// TIA Portal V15.1 export
FUNCTION "CallTemplateTest" : Void   // FC11, LAD
{ S7_Optimized_Access := 'TRUE' }
// stored: SetENOAutomatically False
   VAR_TEMP
      t_PowerRelease : Bool;
   END_VAR
BEGIN

REGION Network 1: Release by power
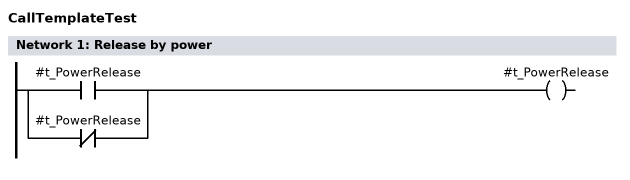
   RUNG wire#powerrail
      Contact( #t_PowerRelease )
      wire#w1
      Coil( #t_PowerRelease )
   END_RUNG
   RUNG wire#powerrail
      I_Contact( #t_PowerRelease )
   END_RUNG wire#w1
   // the same network as SCL:
   #t_PowerRelease := #t_PowerRelease OR NOT #t_PowerRelease;
END_REGION
END_FUNCTION
